// TIA Portal V19 export
DATA_BLOCK "A0302_Manipolatore_PERS"   // DB91
// stored: MemoryReserve 100
   VAR RETAIN
      Par : Struct
         Ax : "Positioning_EPOS_Machine_Par";
         Ax_Aut { S7_SetPoint := 'True'} : "A0301_Mach_Speed_Par";
         Ax_Pos : Struct
            Prelievo { S7_SetPoint := 'True'} : LReal := 0.0;
            BancoCtrl { S7_SetPoint := 'True'} : LReal := -648.0;
            BancoA0303 { S7_SetPoint := 'True'} : LReal := 545.0;
            Tollerance : Struct
               Prelievo { S7_SetPoint := 'True'} : LReal := 1.0;
               BancoCtrl { S7_SetPoint := 'True'} : LReal := 1.0;
               BancoA0303 { S7_SetPoint := 'True'} : LReal := 1.0;
            END_STRUCT;
         END_STRUCT;
      END_STRUCT;
      Pers_Data : Struct
         EncoderAbsolute_Preset_OK : Bool := TRUE;
         Persistent_ActualPosition : LReal := 0.0;
      END_STRUCT;
   END_VAR
BEGIN
   Par.Ax.PosTolerance := 0.5;
   Par.Ax.DelayInPosition := T#500MS;
   Par.Ax.Man_Vel := 10000.0;
   Par.Ax.Man_Acc := 1500.0;
   Par.Ax.Man_Dec := 1500.0;
   Par.Ax_Aut.SemiAut_Vel := 30000.0;
   Par.Ax_Aut.Aut_Vel := 30000.0;
   Par.Ax_Aut.Aut_Acc := 2000.0;
   Par.Ax_Aut.Aut_Dec := 2000.0;
END_DATA_BLOCK
